// A passing test whose cleanup hangs still proved the code correct. The verdict
// stands.
//
// The overrun is reported separately - TeardownOverran, with a diagnostic and the
// label - because the SUITE has to raise a framework error for it and the runner
// holds no reporters. On a rig this may mean an axis left powered, so it must be
// loud without being a lie about the test.
FUNCTION_BLOCK TEST_RunnerTeardownOverrunKeepsTheVerdict IMPLEMENTS I_Test
VAR
	// A private runner, driven one scan per call. The outer test spans scans by
	// returning FALSE, which is exactly the mechanism being verified one level down.
	Registry : TestRegistry<1>;
	Runner	 : TestRunner;
	Handle	 : TestVerdict;
	Budgets	 : ST_TestBudgets;
	Journal	 : REFERENCE TO TestJournal;
	Slot	 : ST_TestSlot;
	Outcome	 : E_PhaseOutcome;
	Loaded	 : BOOL;
	Phase	 : DINT;
	Scans	 : DINT;
	Subject : HangingTeardownTest;

	ExpectedTwo : UDINT;
	ActualCount : UDINT;
	ExpectedStatus : E_TestStatus;
	ActualStatus   : E_TestStatus;
	Diagnostic	   : T_MaxString;
	ActiveLabel	   : T_MaxString;
	ExpectedLabel  : T_MaxString;
END_VAR

METHOD Run : BOOL
VAR_INPUT
	Enable : BOOL;
	Test   : I_TestAssertions;
END_VAR
Scans := Scans + 1;
IF Scans > 200 THEN
	Test.Fail('the subject never reached a terminal outcome');
	Run := TRUE;
	RETURN;
END_IF

CASE Phase OF

0:
	Budgets.Teardown.Cycles		 := 2;
	Budgets.Teardown.IsCyclesSet := TRUE;

	Registry.TryClaim(Subject, 'teardown hangs', Budgets);
	Runner.Attach(Roster := Registry, Verdict := Handle);
	Slot   := Registry.Slot(0);
	Loaded := Runner.Load(Slot);
	Phase   := 1;
	Run	   := FALSE;

1:
	Outcome := Runner.Advance(Enable := TRUE);
	IF Outcome <> E_PhaseOutcome.Running THEN
		// Read before anything else can unload it.
		Diagnostic	:= Runner.TeardownDiagnostic;
		ActiveLabel := Runner.ActiveLabel;
		Phase		:= 2;
	END_IF
	Run := FALSE;

2:
	Test.AssertTrue(Outcome = E_PhaseOutcome.TeardownOverran, 'reported as an overrun');

	ExpectedTwo := 2;
	ActualCount := Subject.TeardownCalls;
	Test.AssertEqual(ExpectedTwo, ActualCount, 'teardown got its own budget');

	Test.AssertTrue(Diagnostic <> '', 'a diagnostic was composed');
	Test.AssertTrue(FIND(Diagnostic, 'teardown') > 0, 'and it names the phase');

	ExpectedLabel := 'teardown hangs';
	Test.AssertEqual(ExpectedLabel, ActiveLabel, 'and the test that hung');

	// The point of the whole test.
	Journal REF= Registry.Journal(0);
	IF __ISVALIDREF(Journal) THEN
		ExpectedStatus := E_TestStatus.Passed;
		ActualStatus   := Journal.Status;
		Test.AssertEqual(ExpectedStatus, ActualStatus, 'the verdict is untouched');
	END_IF

	Run := TRUE;

END_CASE
END_METHOD

END_FUNCTION_BLOCK

(* stored: Version 1.1.0.1, ProductVersion 3.1.4026.18
   POU TEST_RunnerTeardownOverrunKeepsTheVerdict: Id {feeb2e59-b7d0-4d76-9715-38f6e6606e43}, SpecialFunc None
   Folder I_Test: Id {37f3d977-21fb-49e5-afa1-73622ecc0590}
   Method Run: Id {4ff3ec1e-1361-45d0-ab12-c3c0eaffaa56} *)
